INTERFACE I_RpcApi

METHOD CyclicCall
VAR_INPUT
END_VAR
END_METHOD

METHOD RegisterAsynchronousRpcHandlersWith
VAR_INPUT
	Host : I_HostAsynchronousRpcHandlers;
END_VAR
END_METHOD

METHOD RegisterSynchronousRpcHandlersWith
VAR_INPUT
	Host : I_HostSynchronousRpcHandlers;
END_VAR
END_METHOD

END_INTERFACE

(* stored: Version 1.1.0.1, ProductVersion 3.1.4026.13
   Itf I_RpcApi: Id {17b083e7-ae0c-0c94-08dc-e56a38b862e4}
   Method CyclicCall: Id {e1d77c4a-cc84-0af2-1e64-ac22f705b29d}
   Method RegisterAsynchronousRpcHandlersWith: Id {188eb446-b1db-03a5-28d1-127fd6bacf08}
   Method RegisterSynchronousRpcHandlersWith: Id {8ef3eb5f-10d2-0144-240b-5ae24d5edb8e} *)
